{attribute 'qualified_only'}
VAR_GLOBAL
	// Execute flags for vacuum system operations
	{attribute 'pytmc' := '
		pv: PLC_LAS_BTS_VAC:OPERATION:CANCEL
		io: i		
	'}
	i_bCancel : BOOL;
	
	{attribute 'pytmc' := '
		pv: PLC_LAS_BTS_VAC:OPERATION
		io: io
	'}
	iq_eOperation : E_Op;
	
	{attribute 'pytmc' := '
		pv: PLC_LAS_BTS_VAC:OPERATION:TRANSPORT_TUBE
		io: io
	'}
	iq_eTransportTube : E_TransportTube;
	
	{attribute 'pytmc' := '
		pv: PLC_LAS_BTS_VAC:OPERATION:BUSY
		io: o
		field: ZNAM NOT_BUSY
		field: ONAM BUSY
	'}
	q_bBusy : BOOL;
	
	{attribute 'pytmc' := '
		pv: PLC_LAS_BTS_VAC:LASER_OK
		io: o
		field: ZNAM error
		field: ONAM OK
	'}
	q_bLaserOk : BOOL;
	
	{attribute 'pytmc' := '
		pv: PLC_LAS_BTS_VAC:OPERATION:MESSAGE
		io: o
	'}
	q_sMessage : STRING(EPICS_STRING_SIZE);
END_VAR

(* stored: Version 1.1.0.1, ProductVersion 3.1.4022.17
   GVL GVL_Operation: Id {2dd51a79-7824-0563-37ec-bbc7ba082317} *)
